PROGRAM MAIN
VAR
	//updatetimestamparrayobject : ST_Event;
	//flag : Bool := True;
	eEventType : E_EventType:= E_EventType.Alaram;
	eEventSeverity : TcEventseverity := TcEventSeverity.Error;
	nEventIdentity : UDINT := 143;
	sEventText : STRING(255):= 'Testing out how function blocks work';
	
	flag: BOOL := FALSE;
	SaveCSVFile : FB_SaveasCSVFile;
	EventLogger : eventLogger(SaveCSVFile);
END_VAR

IF flag THEN
	EventLogger.AddEvent(eEventType,eEventSeverity,nEventIdentity, sEventText);
	flag:= FALSE;
END_IF

SaveCSVFile();

END_PROGRAM

(* stored: Version 1.1.0.1, ProductVersion 3.1.4024.16
   POU MAIN: Id {84b73be5-16fa-4af9-bcfa-2727274586e4}, SpecialFunc None *)
